{attribute 'GeneratedUsingTerminal: EK1122-0000-0018'}
{attribute addProperty BoxType "EK1122-0000-0018"}
{attribute addProperty Id "Beckhoff_EP6xxxsub_EK1100EK1100_AB5A94672A_0001_EP6001_0002_0020EP6001_B965E9F560A_0002_EP6001_0002_0021EP6001_B965E9F560A_0003_EP6002_0002_0016EP6002_7F9F5532108A_0004_EP6002_0002_0017EP6002_EA7A2404108A_0005_EP6002_0002_0018EP6002_EA7A2404108A_0006_EP6002_0002_0019EP6002_EA7A2404108A_0007_EP6002_0002_0020EP6002_EA7A2404108A_0008_EP6002_0002_0021EP6002_EA7A2404108A_0009_EP6002_0002_0023EP6002_EECF1379108A_0010_EP6002_0002_0024EP6002_EECF1379108A_0011_EP6090_0000_0017EP6090_1BDB3CCC22A_0012_EP6224_0002_0016EP6224_95138EAB28A_0013_EP6224_0042_0016EP6224_9F81C08032A_0014_EP6224_2022_0016EP6224_498F30FB24A_0015_EP6224_2022_0017EP6224_498F30FB24A_0016_EP6224_2022_0018EP6224_9A0D50E824A_0017_EP6224_3022_0016EP6224_498F30FB24A_0018_EP6224_3022_0017EP6224_9A0D50E824A_0019_EP6228_0022_0016EP6228_F9D6B3C628A_0020_EP6228_0022_0017EP6228_F9D6B3C628A_0021_EP6228_0022_0018EP6228_F9D6B3C628A_0022_EP6228_0042_0016EP6228_0C20E27E36A_0023_EP6228_3032_0016EP6228_F9D6B3C628A_0024_EP6228_3132_0016EP6228_877E0FC232A_0025_EP6228_3142_0016EP6228_877E0FC232A_0026_EP6601_0002_0018EP6601_DA9BE95610"}
{attribute addProperty CRC "337247705"}
{attribute addProperty Size "1410"}
TYPE Beckhoff_EP6xxxEK1122_1419FDD9 EXTENDS EK1122_AB5A9467 :
STRUCT
	{attribute addProperty Name "Beckhoff_EP6xxxsub_EK1100"}
	Beckhoff_EP6xxxsub_EK1100 : EK1100_AB5A9467;
	{attribute addProperty Name "A_0001_EP6001_0002_0020"}
	A_0001_EP6001_0002_0020 : EP6001_B965E9F5;
	{attribute addProperty Name "A_0002_EP6001_0002_0021"}
	A_0002_EP6001_0002_0021 : EP6001_B965E9F5;
	{attribute addProperty Name "A_0003_EP6002_0002_0016"}
	A_0003_EP6002_0002_0016 : EP6002_7F9F5532;
	{attribute addProperty Name "A_0004_EP6002_0002_0017"}
	A_0004_EP6002_0002_0017 : EP6002_EA7A2404;
	{attribute addProperty Name "A_0005_EP6002_0002_0018"}
	A_0005_EP6002_0002_0018 : EP6002_EA7A2404;
	{attribute addProperty Name "A_0006_EP6002_0002_0019"}
	A_0006_EP6002_0002_0019 : EP6002_EA7A2404;
	{attribute addProperty Name "A_0007_EP6002_0002_0020"}
	A_0007_EP6002_0002_0020 : EP6002_EA7A2404;
	{attribute addProperty Name "A_0008_EP6002_0002_0021"}
	A_0008_EP6002_0002_0021 : EP6002_EA7A2404;
	{attribute addProperty Name "A_0009_EP6002_0002_0023"}
	A_0009_EP6002_0002_0023 : EP6002_EECF1379;
	{attribute addProperty Name "A_0010_EP6002_0002_0024"}
	A_0010_EP6002_0002_0024 : EP6002_EECF1379;
	{attribute addProperty Name "A_0011_EP6090_0000_0017"}
	A_0011_EP6090_0000_0017 : EP6090_1BDB3CCC;
	{attribute addProperty Name "A_0012_EP6224_0002_0016"}
	A_0012_EP6224_0002_0016 : EP6224_95138EAB;
	{attribute addProperty Name "A_0013_EP6224_0042_0016"}
	A_0013_EP6224_0042_0016 : EP6224_9F81C080;
	{attribute addProperty Name "A_0014_EP6224_2022_0016"}
	A_0014_EP6224_2022_0016 : EP6224_498F30FB;
	{attribute addProperty Name "A_0015_EP6224_2022_0017"}
	A_0015_EP6224_2022_0017 : EP6224_498F30FB;
	{attribute addProperty Name "A_0016_EP6224_2022_0018"}
	A_0016_EP6224_2022_0018 : EP6224_9A0D50E8;
	{attribute addProperty Name "A_0017_EP6224_3022_0016"}
	A_0017_EP6224_3022_0016 : EP6224_498F30FB;
	{attribute addProperty Name "A_0018_EP6224_3022_0017"}
	A_0018_EP6224_3022_0017 : EP6224_9A0D50E8;
	{attribute addProperty Name "A_0019_EP6228_0022_0016"}
	A_0019_EP6228_0022_0016 : EP6228_F9D6B3C6;
	{attribute addProperty Name "A_0020_EP6228_0022_0017"}
	A_0020_EP6228_0022_0017 : EP6228_F9D6B3C6;
	{attribute addProperty Name "A_0021_EP6228_0022_0018"}
	A_0021_EP6228_0022_0018 : EP6228_F9D6B3C6;
	{attribute addProperty Name "A_0022_EP6228_0042_0016"}
	A_0022_EP6228_0042_0016 : EP6228_0C20E27E;
	{attribute addProperty Name "A_0023_EP6228_3032_0016"}
	A_0023_EP6228_3032_0016 : EP6228_F9D6B3C6;
	{attribute addProperty Name "A_0024_EP6228_3132_0016"}
	A_0024_EP6228_3132_0016 : EP6228_877E0FC2;
	{attribute addProperty Name "A_0025_EP6228_3142_0016"}
	A_0025_EP6228_3142_0016 : EP6228_877E0FC2;
	{attribute addProperty Name "A_0026_EP6601_0002_0018"}
	A_0026_EP6601_0002_0018 : EP6601_DA9BE956;
END_STRUCT
END_TYPE

(* stored: Version 1.2.0.0, ProductVersion 3.1.4024.9
   DUT Beckhoff_EP6xxxEK1122_1419FDD9: Id {d699b80f-4b8a-4165-87e1-7bb4179ad495} *)
